{attribute addProperty BoxType "EL2521-0124-0018"}
{attribute addProperty Id "StatusAT %I*Status_66AE5E45162"}
{attribute addProperty CRC "2087802025"}
{attribute addProperty SizeInBites "16"}
{attribute addProperty SizeInBytes "2"}
TYPE PTO_Status_7C7154A9 :
STRUCT
	{attribute addProperty Name "Status"}
	Status AT %I* : Status_66AE5E45;
END_STRUCT
END_TYPE

(* stored: Version 1.2.0.0, ProductVersion 3.1.4024.9
   DUT PTO_Status_7C7154A9: Id {0861275b-5eea-434e-a23e-eec3d1721a39} *)
